FUNCTION_BLOCK OP_Selection (* Composite Function Block Type *)
  (* Standard: 61499-2 *)
  (* Version 0.0, 4/16/2020, prana, nxtControl GmbH, template *)
  PACKAGE Main;
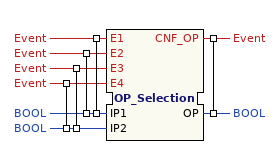
  EVENT_INPUT
    E1 WITH IP1; (* Initialization Request *)
    E2 WITH IP1; (* Normal Execution Request *)
    E3 WITH IP2;
    E4 WITH IP2;
  END_EVENT
  EVENT_OUTPUT
    CNF_OP WITH OP;
  END_EVENT
  VAR_INPUT
    IP1 : BOOL; (* Input event qualifier *)
    IP2 : BOOL;
  END_VAR
  VAR_OUTPUT
    OP : BOOL; (* Output event qualifier *)
  END_VAR
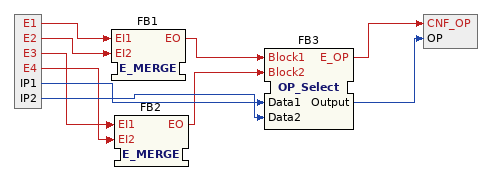
  FBS
    FB1 : E_MERGE;
    FB2 : E_MERGE;
    FB3 : OP_Select;
  END_FBS
  EVENT_CONNECTIONS
    FB3.E_OP TO CNF_OP;
    FB1.EO TO FB3.Block1;
    FB2.EO TO FB3.Block2;
    E1 TO FB1.EI1;
    E2 TO FB1.EI2;
    E3 TO FB2.EI1;
    E4 TO FB2.EI2;
  END_CONNECTIONS
  DATA_CONNECTIONS
    FB3.Output TO OP;
    IP1 TO FB3.Data1;
    IP2 TO FB3.Data2;
  END_CONNECTIONS
END_FUNCTION_BLOCK
